{attribute 'GeneratedUsingTerminal: EL3208-0000-0017'}
{attribute addProperty BoxType "EL3208-0000-0017"}
{attribute addProperty Id "EtcSlaveTerminalBaseRTD_Inputs_Channel_1AT %I*RTD_Inputs_Channel_9575FEA17RTD_Inputs_Channel_2AT %I*RTD_Inputs_Channel_9575FEA17RTD_Inputs_Channel_3AT %I*RTD_Inputs_Channel_9575FEA17RTD_Inputs_Channel_4AT %I*RTD_Inputs_Channel_9575FEA17RTD_Inputs_Channel_5AT %I*RTD_Inputs_Channel_9575FEA17RTD_Inputs_Channel_6AT %I*RTD_Inputs_Channel_9575FEA17RTD_Inputs_Channel_7AT %I*RTD_Inputs_Channel_9575FEA17RTD_Inputs_Channel_8AT %I*RTD_Inputs_Channel_9575FEA17WcStateAT %I*WcState_9091E0EB2InfoDataAT %I*InfoData_32EB74EA10"}
{attribute addProperty CRC "1547558541"}
{attribute addProperty Size "68"}
TYPE EL3208_5C3DDE8D EXTENDS EtcSlaveTerminalBase :
STRUCT
	{attribute addProperty Name "RTD_Inputs_Channel_1"}
	RTD_Inputs_Channel_1 : RTD_Inputs_Channel_9575FEA1;
	{attribute addProperty Name "RTD_Inputs_Channel_2"}
	RTD_Inputs_Channel_2 : RTD_Inputs_Channel_9575FEA1;
	{attribute addProperty Name "RTD_Inputs_Channel_3"}
	RTD_Inputs_Channel_3 : RTD_Inputs_Channel_9575FEA1;
	{attribute addProperty Name "RTD_Inputs_Channel_4"}
	RTD_Inputs_Channel_4 : RTD_Inputs_Channel_9575FEA1;
	{attribute addProperty Name "RTD_Inputs_Channel_5"}
	RTD_Inputs_Channel_5 : RTD_Inputs_Channel_9575FEA1;
	{attribute addProperty Name "RTD_Inputs_Channel_6"}
	RTD_Inputs_Channel_6 : RTD_Inputs_Channel_9575FEA1;
	{attribute addProperty Name "RTD_Inputs_Channel_7"}
	RTD_Inputs_Channel_7 : RTD_Inputs_Channel_9575FEA1;
	{attribute addProperty Name "RTD_Inputs_Channel_8"}
	RTD_Inputs_Channel_8 : RTD_Inputs_Channel_9575FEA1;
	{attribute addProperty Name "WcState"}
	WcState : WcState_9091E0EB;
	{attribute addProperty Name "InfoData"}
	InfoData : InfoData_32EB74EA;
END_STRUCT
END_TYPE

(* stored: Version 1.2.0.0, ProductVersion 3.1.4024.9
   DUT EL3208_5C3DDE8D: Id {f9b1ae83-4951-4b4b-a52f-903a4484aca4} *)
